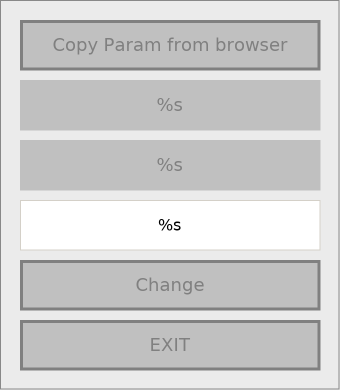
VISUALIZATION ParamDialog  // 340x390
VAR_INPUT
	active_object: I_SYS_COMP_Object;
END_VAR
VAR
	active_param: I_Param;
	name: STRING := 'ParamName';
	value: STRING := 'EnterNewValue';
	actual_value: STRING := 'ParamValue';

END_VAR
    RoundedRectangle (0,0 340x390)
    RoundedRectangle (20,140 300x50), "%s", text variable: actual_value
    RoundedRectangle (20,320 300x50), "EXIT"
        OnMouseUp: CloseDialog Dialog=ParamDialog, Result=OK, NumpadKeypadSet=True
    RoundedRectangle (20,20 300x50), "Copy Param from browser"
        OnMouseUp: execute {
            IF active_object <> 0 THEN
            	active_param := F_IObject_TO_IParam(active_object, active_param);
            	IF active_param <> 0 THEN
            		name := active_param.name;
            		value := active_param.display;
            		actual_value := active_param.display;
            	ELSE
            		name := 'Object is not Param!';
            		value := '';
            		actual_value := '';
            	END_IF
            ELSE
            	name := 'No Object selected!';
            	value := '';
            	actual_value := '';
            END_IF
        }
    Textfield (20,200 300x50), "%s", text variable: value
        OnMouseUp: write the text variable via Default
    RoundedRectangle (20,260 300x50), "Change"
        OnMouseUp: execute {
            IF active_param <> 0 THEN
            	active_param.Change_Param(value);
            	actual_value := active_param.display;
            END_IF
        }
    RoundedRectangle (20,80 300x50), "%s", text variable: name
END_VISUALIZATION

(* stored: Version 1.1.0.1, ProductVersion 3.1.4024.12
   Visu ParamDialog: Id {c850195a-2804-4293-9d51-57de8c90622f} *)
